{attribute 'qualified_only'}
{attribute 'strict'}
TYPE E_Pump_State :
(
	Stopped := 0,
	Starting,
	Runing,
	Error
);
END_TYPE

(* stored: Version 1.1.0.1, ProductVersion 3.1.4024.11
   DUT E_Pump_State: Id {a6c8be50-2caa-49b3-bcc1-412a080fd580} *)
